RoboDK station: 터틀봇이동.rdk

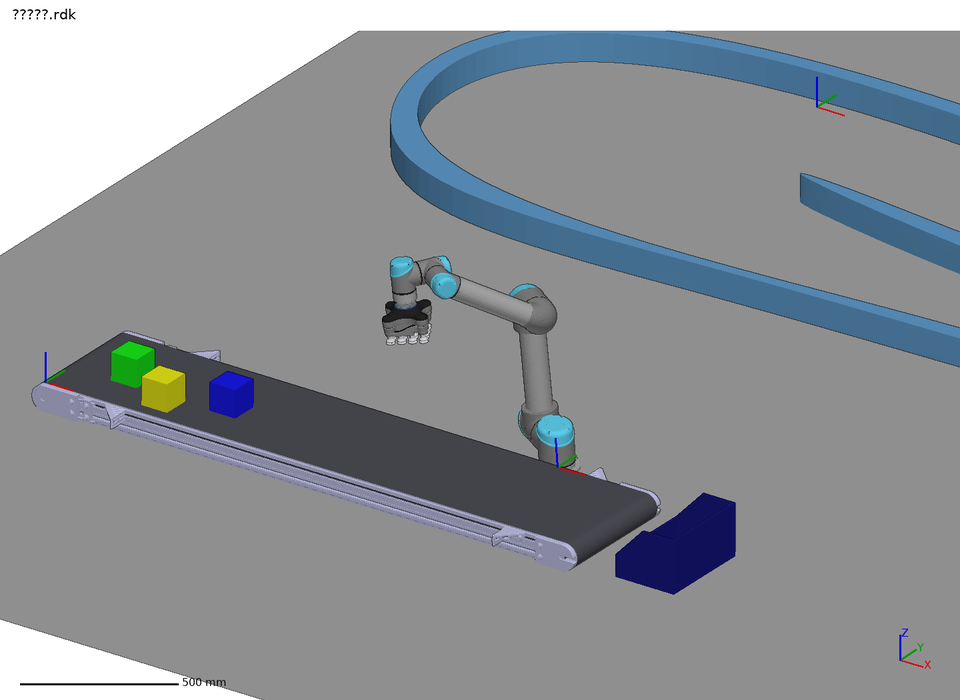
[picture v0: the station drawn from its stored meshes, robots at their saved joint values, targets as dots, program paths as lines]
Station New Station (saved by RoboDK 5.7.4). Poses are relative to the parent item; angles as X-Y-Z fixed-axis rotations.
  - frame MainFrame at (0, 0, 0) mm
  - frame UR5 Base at (820, -2600, 0) mm, rotated rx 1.76 ry -2.58 rz 0 deg
    - robot UR5: 6 axes
        modified DH rows (alpha deg, a mm, theta deg, d mm): 0, 0, 0, 89.2; 90, 0, 180, 0; 0, 425, 0, 0; 0, 392, 0, 109.3; -90, 0, 0, 94.75; 90, 0, 180, 82.5
        joint limits [-360, -360, -360, -360, -360, -360] to [360, 360, 360, 360, 360, 360]; home [0, -90, -90, 0, 90, 0]; saved at [-124.91, -91.831, -55.836, -123.799, 93.237, -64.705]
      - tool OnRobot VG10 Vacuum Gripper, TCP at (0, 0, 130.9) mm, size 145.4 x 145.4 x 118.3 mm
  - object Floor at (0, -3000, 0) mm, size 3000 x 3000 x 0 mm, geometry from Floor (1).sld
  - object Floor at (3000, -3000, 0) mm, size 3000 x 3000 x 0 mm, geometry from Floor (1).sld
  - object Floor at (0, 0, 0) mm, size 3000 x 3000 x 0 mm, geometry from Floor (1).sld
  - object Floor at (3000, 0, 0) mm, size 3000 x 3000 x 0 mm, geometry from Floor (1).sld
  - object Bin Red at (2930, 150, 0) mm, rotated rx 0 ry 0 rz -180 deg, size 225 x 337.5 x 191.2 mm, geometry from Bin-Red.sld
  - object Bin Blue at (1420, -2800, 0) mm, rotated rx 0 ry 0 rz -180 deg, size 225 x 337.5 x 191.2 mm, geometry from Bin-Blue.sld
  - object path at (5000, -200, 0) mm, size 3159.6 x 1446.5 x 100 mm, geometry from path.step
  - object path2 at (-2520, -560, 40) mm, rotated rx 0 ry 0 rz 180 deg, size 3159.6 x 1446.5 x 100 mm, geometry from path.step
  - object Yellow at (-350, -3100, 100) mm, size 100 x 100 x 100 mm, geometry from Yellow.step
  - object Green at (-530, -3010, 100) mm, size 100 x 100 x 100 mm, geometry from Green.step
  - object Blue at (-150, -3010, 100) mm, size 100 x 100 x 100 mm, geometry from Blue.step
  - frame Conveyor Belt (2m) Base at (-740, -3190, 100) mm
    - robot Conveyor Belt (2m): 1 axes
        modified DH rows (alpha deg, a mm, theta deg, d mm): 0, 0, 0, 0 linear
        base shift (0, 0, 0) mm, rotated rx 0 ry 90 rz 0 deg
        joint limits [-500000] to [500000]; home [0]; saved at [0]
  - frame turtlebot Base at (2640, -20, 20) mm
    - object turtlebot3_waffle (1) at (0, 0, 0) mm, size 280.7 x 305.1 x 138.1 mm, geometry from turtlebot3_waffle (1).step
    - object Red at (0, -90, 90) mm, size 100 x 100 x 100 mm, geometry from Red.step
  - Python program Prog1 (listed below)
  - frame Frame 1 at (0, 1500, 20) mm

--- Python program Prog1 ---
from robodk import robolink
from robodk.robomath import *
import time
import math

RDK = robolink.Robolink()

# =========================
# RoboDK 아이템 이름
# =========================
turtle_base = RDK.Item("turtlebot Base")
red_box = RDK.Item("Red")

if not turtle_base.Valid():
    raise Exception("turtlebot Base를 찾을 수 없습니다. 이름을 확인하세요.")

# =========================
# 시작 위치 + 경유지 좌표
# [X, Y, Z]
# =========================
START = [1210, -2510, 20]

WAYPOINTS = [
    [2560, -1140, 20],   # Frame 5
    [-340, -780, 20],    # Frame 4
    [330, -380, 20],     # Frame 3
    [1960, -450, 20],    # Frame 2
    [2640, -20, 20],     # Frame 1
]

# =========================
# Red 박스를 터틀봇에 붙이기
# =========================
if red_box.Valid():
    red_abs_pose = red_box.PoseAbs()
    red_box.setParentStatic(turtle_base)
    red_box.setPoseAbs(red_abs_pose)
    print("Red 박스를 turtlebot Base에 붙였습니다.")
else:
    print("Red 박스를 찾지 못했습니다. 박스 없이 이동합니다.")

# =========================
# pose 생성 함수
# =========================
def make_pose(x, y, z, yaw_deg=0):
    """
    x, y, z 위치와 z축 회전각으로 RoboDK pose 생성
    yaw_deg: 터틀봇 방향 각도
    """
    return transl(x, y, z) * rotz(math.radians(yaw_deg))

# =========================
# 두 점 사이 방향각 계산
# =========================
def calc_yaw_deg(p1, p2):
    dx = p2[0] - p1[0]
    dy = p2[1] - p1[1]
    return math.degrees(math.atan2(dy, dx))

# =========================
# 부드러운 이동 함수
# =========================
def move_smooth(item, target_pose, speed=350, dt=0.03):
    start_pose = item.PoseAbs()

    start = Pose_2_TxyzRxyz(start_pose)
    target = Pose_2_TxyzRxyz(target_pose)

    dx = target[0] - start[0]
    dy = target[1] - start[1]
    dist = math.sqrt(dx * dx + dy * dy)

    steps = max(1, int(dist / (speed * dt)))

    for i in range(1, steps + 1):
        ratio = i / steps

        now = [
            start[j] + (target[j] - start[j]) * ratio
            for j in range(6)
        ]

        item.setPoseAbs(TxyzRxyz_2_Pose(now))
        RDK.Render()
        time.sleep(dt)

# =========================
# 실행
# =========================

# 1. 시작 위치로 세팅
start_yaw = calc_yaw_deg(START, WAYPOINTS[0])
turtle_base.setPoseAbs(make_pose(START[0], START[1], START[2], start_yaw))
RDK.Render()
time.sleep(0.5)

print("TurtleBot 이동 시작")

# 2. 경유지 순서대로 이동
current = START

for idx, wp in enumerate(WAYPOINTS):
    yaw = calc_yaw_deg(current, wp)
    target_pose = make_pose(wp[0], wp[1], wp[2], 0)

    print(f"Moving to Frame {5 - idx}: X={wp[0]}, Y={wp[1]}, Z={wp[2]}, Yaw={yaw:.1f}")
    move_smooth(turtle_base, target_pose, speed=350)

    current = wp

print("TurtleBot 이동 완료")
